(* IEC 61131-3 sources: AXOpen/src/templates.simple/app/src/templates/starterunit/DataManagers, 1 file *)

(* ---- FragmentsProcessDataManager.st ---- *)
NAMESPACE axosimple.StarterUnitTemplate
    USING axosimple;
    USING AXOpen.Data;
    USING AXOpen.Core;
    USING System.Strings;

    CLASS FragmentProcessDataManger
        EXTENDS AXOpen.Data.AxoDataExchange
        VAR PUBLIC
            {#ix-generic:TOnline}
            {#ix-generic:TPlain as POCO}
            {#ix-attr:[AXOpen.Data.AxoDataEntityAttribute]}
            {#ix-attr:[Container(Layout.Stack)]}
            Payload : ProcessData;
        END_VAR
    END_CLASS
END_NAMESPACE
